// TIA Portal project "Pilot_Ultrafilter" (V20)

(* hardware
DEVICE "S7-1200 station_1"  S7-1200 Station
   slot 0: "Rack_0"  S7-1200 Rack  Rack  V1.0
   slot 1: "PLC_1"  CPU 1214C DC/DC/Rly  6ES7 214-1HG40-0XB0  V4.5
   slot 2: "AI 8x13BIT_1"  SM 1231 AI8  6ES7 231-4HF32-0XB0  V2.1
   slot 3: "AQ 2x14BIT_1"  SM 1232 AQ2  6ES7 232-4HB32-0XB0  V2.0
*)

// ===== PLC "PLC_1"  CPU 1214C DC/DC/Rly =====

VAR_GLOBAL   // PLC tag table "Default tag table"
   "IT_Pump_DryRun_Fault" AT %M0.0 : Bool;
   "IT_Pump_Wrong_Valve_Setting_fault" AT %M0.1 : Bool;
   "PID_Reset_Value" AT %M0.2 : Bool;
   "IT_EStop_NOk" AT %M0.3 : Bool;
   "ErrorBit" AT %M0.4 : Bool;   // Mindaddig amíg a hiba nem kerül nyugtázásra addig nem lehet elindítani a rendszert
   "Tag_7" AT %M0.5 : Bool;
   "Tag_8" AT %M0.6 : Bool;
   "Tag_9" AT %M0.7 : Bool;
   "Tag_10" AT %M1.0 : Bool;
   "Tag_11" AT %M1.1 : Bool;
   "Tag_12" AT %M1.2 : Bool;
   "Clock_Byte" AT %MB10 : Byte;
   "Clock_10Hz" AT %M10.0 : Bool;
   "Clock_5Hz" AT %M10.1 : Bool;
   "Clock_2.5Hz" AT %M10.2 : Bool;
   "Clock_2Hz" AT %M10.3 : Bool;
   "Clock_1.25Hz" AT %M10.4 : Bool;
   "Clock_1Hz" AT %M10.5 : Bool;
   "Clock_0.625Hz" AT %M10.6 : Bool;
   "Clock_0.5Hz" AT %M10.7 : Bool;
END_VAR

VAR_GLOBAL   // PLC tag table "Digital_Inputs"
   "DI_EStop_Ok" AT %I0.0 : Bool;   // VészStop alaphelyzetben NC
   "DI_MotorProtectionSwitch" AT %I0.1 : Bool;   // Motorvédő kapcsoló NC
   "DI_TankLevelSwitch" AT %I0.2 : Bool;   // Tartály szintjelző; Üres: 1 ; Tele:0
END_VAR

VAR_GLOBAL   // PLC tag table "Digital Outputs"
   "DO_MotorStartSign" AT %Q0.0 : Bool;
   "DO_TankFillValve" AT %Q0.1 : Bool;
   "DO_OpenPermeateValve" AT %Q0.2 : Bool;
   "DO_GreenLamp" AT %Q0.5 : Bool;
   "DO_RedLamp" AT %Q0.7 : Bool;
END_VAR

VAR_GLOBAL   // PLC tag table "Analog_Inputs"
   "AI_FT01_FlowMeter" AT %IW96 : Int;   // Szivattyú utáni áramlásmérő
   "AI_FT02_FlowMeter" AT %IW98 : Int;   // Permeátum ágban lévő áramlásmérő
   "AI_PT01_PressureTransmitter" AT %IW100 : Int;   // Membrán elötti nyomástávadó
   "AI_PT02_PressureTransmitter" AT %IW102 : Int;   // Membrán utáni nyomástávadó
END_VAR

VAR_GLOBAL   // PLC tag table "Analog_Outputs"
   "AO_PumpSpeed" AT %QW112 : Int;   // Szivattyú fordulatszámának szabályozására való analóg kimenet
END_VAR

// folder: HMI_DataBlocks

DATA_BLOCK "HMI_Inputs"   // DB4
{ S7_Optimized_Access := 'FALSE' }
VERSION : 0.1
   VAR
      "FT01_FlowMeter_l/min" : Real;
      "FT02_FlowMeter_l/min" : Real;
      PT01_PressureTransmitter_bar : Real;
      PT02_PressureTransmitter_bar : Real;
      "P01_PumpPerformance_%" : Real;
   END_VAR
BEGIN
END_DATA_BLOCK

DATA_BLOCK "HMI_Outputs"   // DB5
{ S7_Optimized_Access := 'FALSE' }
VERSION : 0.1
   VAR
      Asked_Total_Flow : Int;
      Asked_Permeate_Flow : Real;
      askedFlushingTime : DInt;
      askedVentingTime : DInt;
      "askedPumpPerformance_%" : Int;
      askedState : Int;
      askedPermeateFlowMonitoring : Bool;
      Motor_Start_Sign : Bool;
      Nyugta : Bool;
      askedGreenLight : Bool;
      askedRedLight : Bool;
      askedTankFillValveOpen : Bool;
      askedPermeateValveOpen : Bool;
   END_VAR
BEGIN
END_DATA_BLOCK

// folder: Internal_DataBlocks

DATA_BLOCK "DB_AnalogCalculatedValues"   // DB2
{ S7_Optimized_Access := 'TRUE' }
VERSION : 0.1
   VAR
      "FT01_FlowMeter_l/min" : Real;
      "FT02_FlowMeter_l/min" : Real;
      PT01_PressureTransmitter_bar : Real;
      PT02_PressureTransmitter_bar : Real;
      "P01_PumpPerformance_%" : Real;
   END_VAR
BEGIN
END_DATA_BLOCK

DATA_BLOCK "FB_ErrorHandler_DB_1"   // DB9
{ S7_Optimized_Access := 'TRUE' }
VERSION : 0.1
// stored: InstanceOfName FB_ErrorHandler
"FB_ErrorHandler"
BEGIN
END_DATA_BLOCK

DATA_BLOCK "FB_ErrorHandler_DB"   // DB10
{ S7_Optimized_Access := 'TRUE' }
VERSION : 0.1
// stored: InstanceOfName FB_ErrorHandler
"FB_ErrorHandler"
BEGIN
END_DATA_BLOCK

DATA_BLOCK "DB_StateMachine"   // DB11
{ S7_Optimized_Access := 'FALSE' }
VERSION : 0.1
   VAR
      actualState : Int;
      initState : Int := 0;
      idleState : Int := 10;
      serviceState : Int := 20;
      filteringState : Int := 100;
      filteringStateTankFilling : Int := 110;
      filteringStateVenting : Int := 120;
      filteringStateFiltering : Int := 130;
      filteringStateFlushing : Int := 140;
      filteringEnded : Int := 200;
      errorState : Int := 900;
      initState_bool : Bool;
      idleState_bool : Bool;
      serviceState_bool : Bool;
      filteringState_bool : Bool;
      filteringStateTankFilling_bool : Bool;
      filteringStateVenting_bool : Bool;
      filteringStateFiltering_bool : Bool;
      filteringStateFlushing_bool : Bool;
      filteringEnded_bool : Bool;
      errorState_bool : Bool;
   END_VAR
BEGIN
END_DATA_BLOCK

DATA_BLOCK "DB_Errors&Warnings"   // DB12
{ S7_Optimized_Access := 'FALSE' }
VERSION : 0.1
   VAR
      error : Bool;
      warning : Bool;
   END_VAR
BEGIN
END_DATA_BLOCK

DATA_BLOCK "FB_ErrorHandler_DB_2"   // DB17
{ S7_Optimized_Access := 'TRUE' }
VERSION : 0.1
// stored: InstanceOfName FB_ErrorHandler
"FB_ErrorHandler"
BEGIN
END_DATA_BLOCK

// folder: System blocks/Program resources

DATA_BLOCK "IEC_Timer_0_DB_4"   // DB13
{ S7_Optimized_Access := 'TRUE' }
AUTHOR : Simatic
FAMILY : IEC
NAME : IEC_TMR
VERSION : 1.0
// stored: InstanceOfName IEC_TIMER
"IEC_TIMER"
BEGIN
END_DATA_BLOCK

DATA_BLOCK "IEC_Timer_0_DB_5"   // DB14
{ S7_Optimized_Access := 'TRUE' }
AUTHOR : Simatic
FAMILY : IEC
NAME : IEC_TMR
VERSION : 1.0
// stored: InstanceOfName IEC_TIMER
"IEC_TIMER"
BEGIN
END_DATA_BLOCK

DATA_BLOCK "IEC_Timer_0_DB_6"   // DB15
{ S7_Optimized_Access := 'TRUE' }
AUTHOR : Simatic
FAMILY : IEC
NAME : IEC_TMR
VERSION : 1.0
// stored: InstanceOfName IEC_TIMER
"IEC_TIMER"
BEGIN
END_DATA_BLOCK

DATA_BLOCK "IEC_Timer_0_DB_7"   // DB16
{ S7_Optimized_Access := 'TRUE' }
AUTHOR : Simatic
FAMILY : IEC
NAME : IEC_TMR
VERSION : 1.0
// stored: InstanceOfName IEC_TIMER
"IEC_TIMER"
BEGIN
END_DATA_BLOCK

// folder: FC's

FUNCTION_BLOCK "FB_ErrorHandler"   // FB1, LAD
{ S7_Optimized_Access := 'TRUE' }
VERSION : 0.1
   VAR_INPUT
      startSign : Bool;
   END_VAR
   VAR
      DryRunTimer : TON_TIME;
      WrongValveSettingTimer : TON_TIME;
   END_VAR
   VAR CONSTANT
      Required_Minimum_Flow : Real := 15.0;
      Maximum_Pressure : Real := 10.0;
   END_VAR
BEGIN

REGION Network 1
   // Szárazonfutás elleni védelem
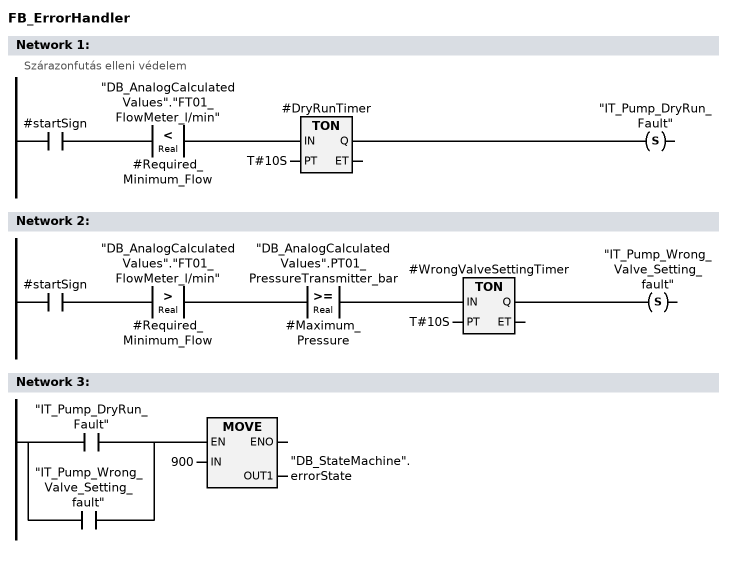
   #DryRunTimer(IN := #startSign AND ("DB_AnalogCalculatedValues"."FT01_FlowMeter_l/min" < #Required_Minimum_Flow),   // TON
                PT := T#10S);
   IF #DryRunTimer.Q THEN "IT_Pump_DryRun_Fault" := TRUE; END_IF;
END_REGION

REGION Network 2
   #WrongValveSettingTimer(IN := #startSign AND ("DB_AnalogCalculatedValues"."FT01_FlowMeter_l/min" > #Required_Minimum_Flow) AND ("DB_AnalogCalculatedValues".PT01_PressureTransmitter_bar >= #Maximum_Pressure),   // TON
                           PT := T#10S);
   IF #WrongValveSettingTimer.Q THEN "IT_Pump_Wrong_Valve_Setting_fault" := TRUE; END_IF;
END_REGION

REGION Network 3
   RUNG wire#powerrail
      Contact( "IT_Pump_DryRun_Fault" )
      wire#w1
      Move(in := 900, out1 => "DB_StateMachine".errorState)
   END_RUNG
   RUNG wire#powerrail
      Contact( "IT_Pump_Wrong_Valve_Setting_fault" )
   END_RUNG wire#w1
   // the same network as SCL:
   IF "IT_Pump_DryRun_Fault" OR "IT_Pump_Wrong_Valve_Setting_fault" THEN
       "DB_StateMachine".errorState := 900;
   END_IF;
END_REGION
END_FUNCTION_BLOCK

FUNCTION "FC_AnalogInputScale" : Void   // FC1, LAD
{ S7_Optimized_Access := 'TRUE' }
VERSION : 0.1
   VAR_INPUT
      InputAnalogValue : Int;
      MinimumAnalogValue : Int;
      MaximumAnalogValue : Int;
      MinimumScaledValue : Real;
      MaxmimumScaledValue : Int;
   END_VAR
   VAR_OUTPUT
      OutputScaledValue : Real;
   END_VAR
   VAR_TEMP
      NormalizedValue : Real;
   END_VAR
BEGIN

REGION Network 1
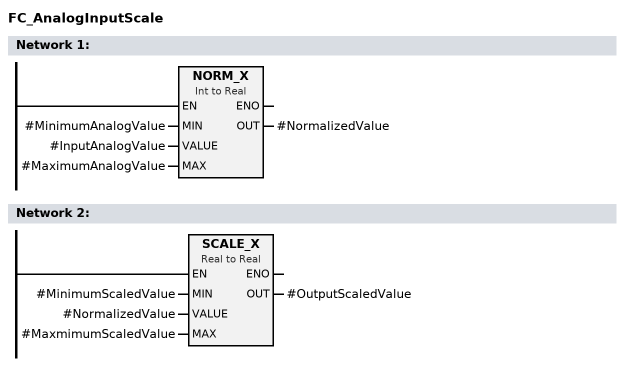
   RUNG wire#powerrail
      { S7_Templates := "[SrcType := Int, DestType := Real]" } Normalize(min := #MinimumAnalogValue, value := #InputAnalogValue, max := #MaximumAnalogValue, out => #NormalizedValue)
   END_RUNG
   // the same network as SCL:
   #NormalizedValue := NORM_X(MIN := #MinimumAnalogValue, VALUE := #InputAnalogValue, MAX := #MaximumAnalogValue);
END_REGION

REGION Network 2
   RUNG wire#powerrail
      { S7_Templates := "[SrcType := Real, DestType := Real]" } Scale(min := #MinimumScaledValue, value := #NormalizedValue, max := #MaxmimumScaledValue, out => #OutputScaledValue)
   END_RUNG
   // the same network as SCL:
   #OutputScaledValue := SCALE_X(MIN := #MinimumScaledValue, VALUE := #NormalizedValue, MAX := #MaxmimumScaledValue);
END_REGION
END_FUNCTION

FUNCTION "FC_ProcessAnalogInputs" : Void   // FC2, LAD
{ S7_Optimized_Access := 'TRUE' }
VERSION : 0.1
   VAR CONSTANT
      FT01_MinimumAnalogValue : Int := 1659;   // Minimális analóg érték a szivattyú utáni áramlásmérő által
      FT02_MinimumAnalogValue : Int := 1382;   // Minimális analóg érték a permeátum ágban lévő áramlásmérőnél
      "PT01-02_MinimumAnalogValue" : Int := 0;   // Minimális analóg érték a két nyomástávadónál
      ALL_MaximumAnalogValue : Int := 27648;   // Maximális analóg érték, összesnél megegyezik
      FT01_MinimumFlowValue : Real := 9.0;   // Legkisebb áramlás amit a szivattyú utáni áramlásmérő tud
      FT02_MinimumFlowValue : Real := 0.5;   // Legkisebb áramlás amit a permeátum ágban lévő áramlásmérő mérni tud
      FT01_MaximumFlowValue : Int := 150;   // Legnagyobb áramlás amit a szivattyú utáni áramlásmérő tud
      FT02_MaximumFlowValue : Int := 10;   // Legnagyobb áramlás amit a premátum ágban lévő áramlásmérő tud
      "PT01-02_MinimumPressureValue" : Real := 0.0;   // Legkisebb nyomás amit a nyomástávadók tudnak
      "PT01-02MaximumPressureValue" : Int := 10;   // Legnagyobb nyomás amit a nyomástávadók tudnak
   END_VAR
   VAR_TEMP   // added for the SCL form of the ladder/FBD networks
      _w1 : Bool;
   END_VAR
BEGIN

REGION Network 1
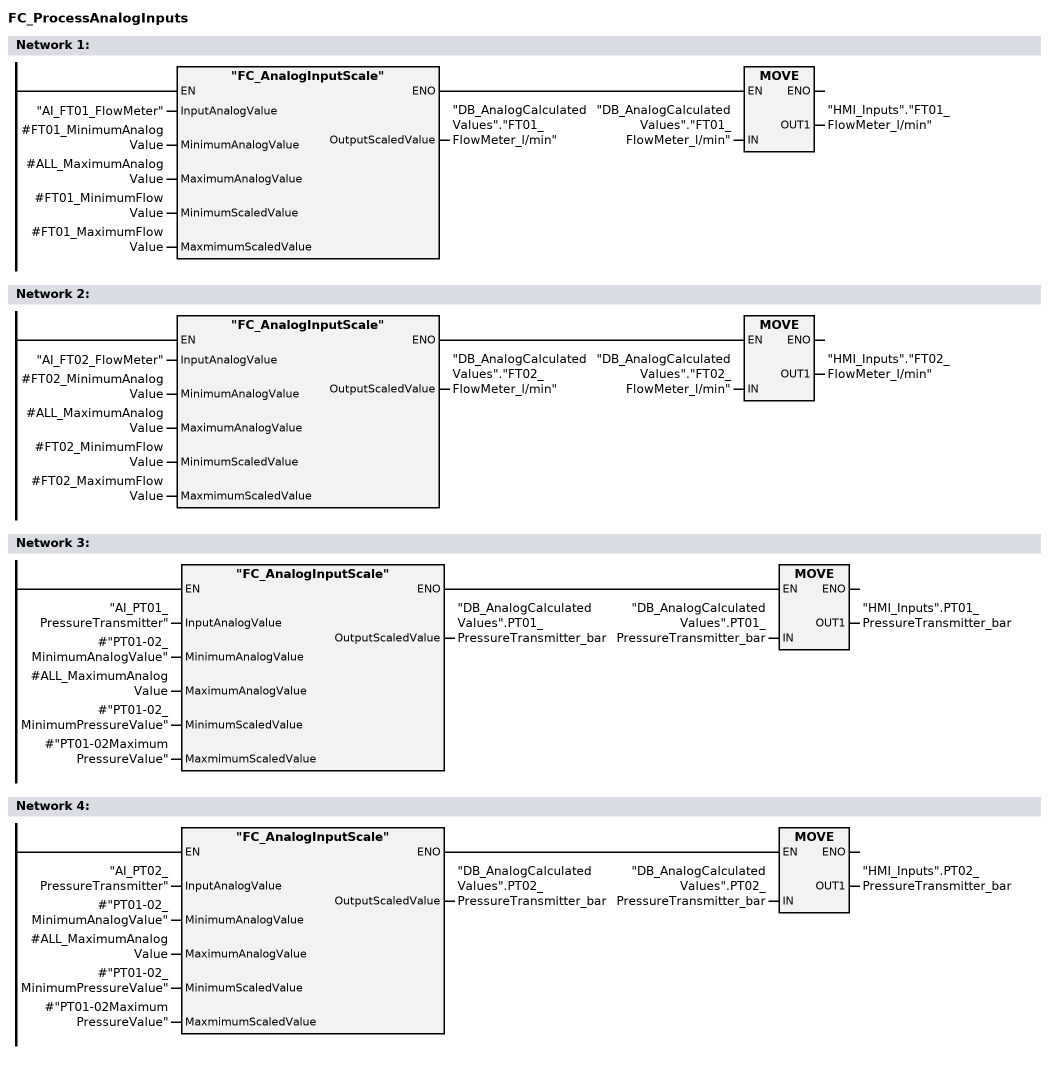
   RUNG wire#powerrail
      "FC_AnalogInputScale"(InputAnalogValue := "AI_FT01_FlowMeter", MinimumAnalogValue := #FT01_MinimumAnalogValue, MaximumAnalogValue := #ALL_MaximumAnalogValue, MinimumScaledValue := #FT01_MinimumFlowValue, MaxmimumScaledValue := #FT01_MaximumFlowValue, OutputScaledValue => "DB_AnalogCalculatedValues"."FT01_FlowMeter_l/min")
      Move(in := "DB_AnalogCalculatedValues"."FT01_FlowMeter_l/min", out1 => "HMI_Inputs"."FT01_FlowMeter_l/min")
   END_RUNG
   // the same network as SCL:
   "FC_AnalogInputScale"(InputAnalogValue := "AI_FT01_FlowMeter",
                         MinimumAnalogValue := #FT01_MinimumAnalogValue,
                         MaximumAnalogValue := #ALL_MaximumAnalogValue,
                         MinimumScaledValue := #FT01_MinimumFlowValue,
                         MaxmimumScaledValue := #FT01_MaximumFlowValue,
                         OutputScaledValue => "DB_AnalogCalculatedValues"."FT01_FlowMeter_l/min",
                         ENO => #_w1);
   IF #_w1 THEN
       "HMI_Inputs"."FT01_FlowMeter_l/min" := "DB_AnalogCalculatedValues"."FT01_FlowMeter_l/min";
   END_IF;
END_REGION

REGION Network 2
   RUNG wire#powerrail
      "FC_AnalogInputScale"(InputAnalogValue := "AI_FT02_FlowMeter", MinimumAnalogValue := #FT02_MinimumAnalogValue, MaximumAnalogValue := #ALL_MaximumAnalogValue, MinimumScaledValue := #FT02_MinimumFlowValue, MaxmimumScaledValue := #FT02_MaximumFlowValue, OutputScaledValue => "DB_AnalogCalculatedValues"."FT02_FlowMeter_l/min")
      Move(in := "DB_AnalogCalculatedValues"."FT02_FlowMeter_l/min", out1 => "HMI_Inputs"."FT02_FlowMeter_l/min")
   END_RUNG
   // the same network as SCL:
   "FC_AnalogInputScale"(InputAnalogValue := "AI_FT02_FlowMeter",
                         MinimumAnalogValue := #FT02_MinimumAnalogValue,
                         MaximumAnalogValue := #ALL_MaximumAnalogValue,
                         MinimumScaledValue := #FT02_MinimumFlowValue,
                         MaxmimumScaledValue := #FT02_MaximumFlowValue,
                         OutputScaledValue => "DB_AnalogCalculatedValues"."FT02_FlowMeter_l/min",
                         ENO => #_w1);
   IF #_w1 THEN
       "HMI_Inputs"."FT02_FlowMeter_l/min" := "DB_AnalogCalculatedValues"."FT02_FlowMeter_l/min";
   END_IF;
END_REGION

REGION Network 3
   RUNG wire#powerrail
      "FC_AnalogInputScale"(InputAnalogValue := "AI_PT01_PressureTransmitter", MinimumAnalogValue := #"PT01-02_MinimumAnalogValue", MaximumAnalogValue := #ALL_MaximumAnalogValue, MinimumScaledValue := #"PT01-02_MinimumPressureValue", MaxmimumScaledValue := #"PT01-02MaximumPressureValue", OutputScaledValue => "DB_AnalogCalculatedValues".PT01_PressureTransmitter_bar)
      Move(in := "DB_AnalogCalculatedValues".PT01_PressureTransmitter_bar, out1 => "HMI_Inputs".PT01_PressureTransmitter_bar)
   END_RUNG
   // the same network as SCL:
   "FC_AnalogInputScale"(InputAnalogValue := "AI_PT01_PressureTransmitter",
                         MinimumAnalogValue := #"PT01-02_MinimumAnalogValue",
                         MaximumAnalogValue := #ALL_MaximumAnalogValue,
                         MinimumScaledValue := #"PT01-02_MinimumPressureValue",
                         MaxmimumScaledValue := #"PT01-02MaximumPressureValue",
                         OutputScaledValue => "DB_AnalogCalculatedValues".PT01_PressureTransmitter_bar,
                         ENO => #_w1);
   IF #_w1 THEN
       "HMI_Inputs".PT01_PressureTransmitter_bar := "DB_AnalogCalculatedValues".PT01_PressureTransmitter_bar;
   END_IF;
END_REGION

REGION Network 4
   RUNG wire#powerrail
      "FC_AnalogInputScale"(InputAnalogValue := "AI_PT02_PressureTransmitter", MinimumAnalogValue := #"PT01-02_MinimumAnalogValue", MaximumAnalogValue := #ALL_MaximumAnalogValue, MinimumScaledValue := #"PT01-02_MinimumPressureValue", MaxmimumScaledValue := #"PT01-02MaximumPressureValue", OutputScaledValue => "DB_AnalogCalculatedValues".PT02_PressureTransmitter_bar)
      Move(in := "DB_AnalogCalculatedValues".PT02_PressureTransmitter_bar, out1 => "HMI_Inputs".PT02_PressureTransmitter_bar)
   END_RUNG
   // the same network as SCL:
   "FC_AnalogInputScale"(InputAnalogValue := "AI_PT02_PressureTransmitter",
                         MinimumAnalogValue := #"PT01-02_MinimumAnalogValue",
                         MaximumAnalogValue := #ALL_MaximumAnalogValue,
                         MinimumScaledValue := #"PT01-02_MinimumPressureValue",
                         MaxmimumScaledValue := #"PT01-02MaximumPressureValue",
                         OutputScaledValue => "DB_AnalogCalculatedValues".PT02_PressureTransmitter_bar,
                         ENO => #_w1);
   IF #_w1 THEN
       "HMI_Inputs".PT02_PressureTransmitter_bar := "DB_AnalogCalculatedValues".PT02_PressureTransmitter_bar;
   END_IF;
END_REGION
END_FUNCTION

FUNCTION "FC_IdleState" : Void   // FC3, SCL
{ S7_Optimized_Access := 'TRUE' }
VERSION : 0.1
BEGIN
   "DO_MotorStartSign" := FALSE;
   "DO_TankFillValve" := FALSE;
   "DO_OpenPermeateValve" := FALSE;
   "DO_GreenLamp" := FALSE;
   "DO_RedLamp" := FALSE;
   "AO_PumpSpeed" := 0;
END_FUNCTION

FUNCTION "FC_TankFilling" : Void   // FC4, LAD
{ S7_Optimized_Access := 'TRUE' }
VERSION : 0.1
BEGIN

REGION Network 1
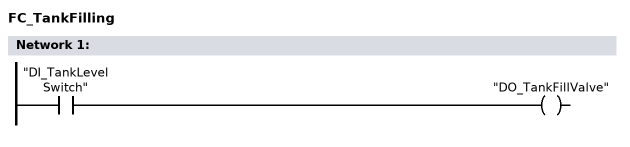
   RUNG wire#powerrail
      Contact( "DI_TankLevelSwitch" )
      Coil( "DO_TankFillValve" )
   END_RUNG
   // the same network as SCL:
   "DO_TankFillValve" := "DI_TankLevelSwitch";
END_REGION
END_FUNCTION

FUNCTION "FC_Membrane_FlushState" : Void   // FC5, LAD
{ S7_Optimized_Access := 'TRUE' }
VERSION : 0.1
   VAR_OUTPUT
      flushingOver : Bool;
      successfullFlushing : Bool;
   END_VAR
   VAR_TEMP
      flushingOverTemp : Bool;
   END_VAR
BEGIN

REGION Network 1
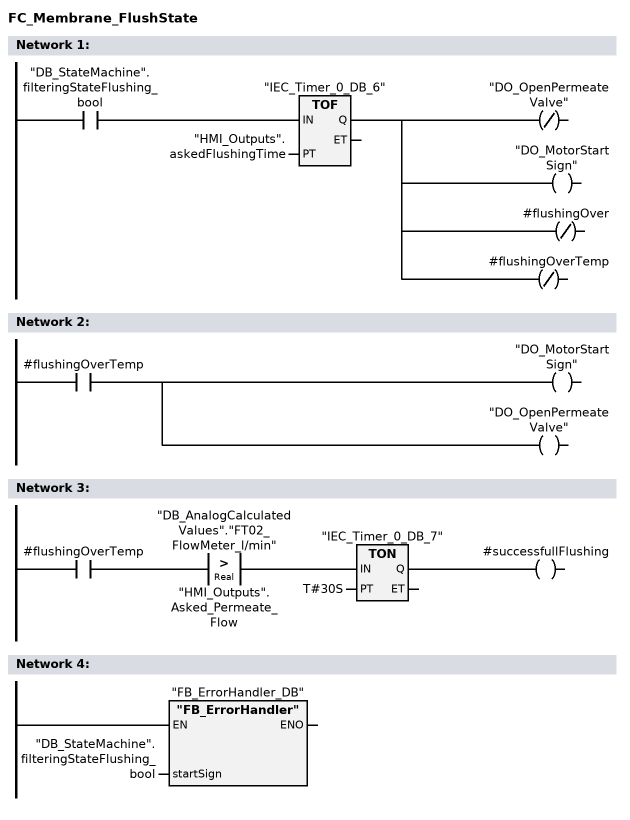
   "IEC_Timer_0_DB_6".TOF(IN := "DB_StateMachine".filteringStateFlushing_bool,
                          PT := "HMI_Outputs".askedFlushingTime);
   "DO_OpenPermeateValve" := NOT "IEC_Timer_0_DB_6".Q;
   "DO_MotorStartSign" := "IEC_Timer_0_DB_6".Q;
   #flushingOver := NOT "IEC_Timer_0_DB_6".Q;
   #flushingOverTemp := NOT "IEC_Timer_0_DB_6".Q;
END_REGION

REGION Network 2
   RUNG wire#powerrail
      Contact( #flushingOverTemp )
      wire#w1
      Coil( "DO_MotorStartSign" )
   END_RUNG
   RUNG wire#w1
      Coil( "DO_OpenPermeateValve" )
   END_RUNG
   // the same network as SCL:
   "DO_MotorStartSign" := #flushingOverTemp;
   "DO_OpenPermeateValve" := #flushingOverTemp;
END_REGION

REGION Network 3
   "IEC_Timer_0_DB_7".TON(IN := #flushingOverTemp AND ("DB_AnalogCalculatedValues"."FT02_FlowMeter_l/min" > "HMI_Outputs".Asked_Permeate_Flow),
                          PT := T#30S);
   #successfullFlushing := "IEC_Timer_0_DB_7".Q;
END_REGION

REGION Network 4
   RUNG wire#powerrail
      "FB_ErrorHandler_DB"(startSign := "DB_StateMachine".filteringStateFlushing_bool)
   END_RUNG
   // the same network as SCL:
   "FB_ErrorHandler_DB"(startSign := "DB_StateMachine".filteringStateFlushing_bool);   // "FB_ErrorHandler"
END_REGION
END_FUNCTION

FUNCTION "FC_ServiceState" : Void   // FC6, LAD
{ S7_Optimized_Access := 'TRUE' }
VERSION : 0.1
// manuális szervíz állás, minden paraméter a HMI ről állítható
BEGIN

REGION Network 1
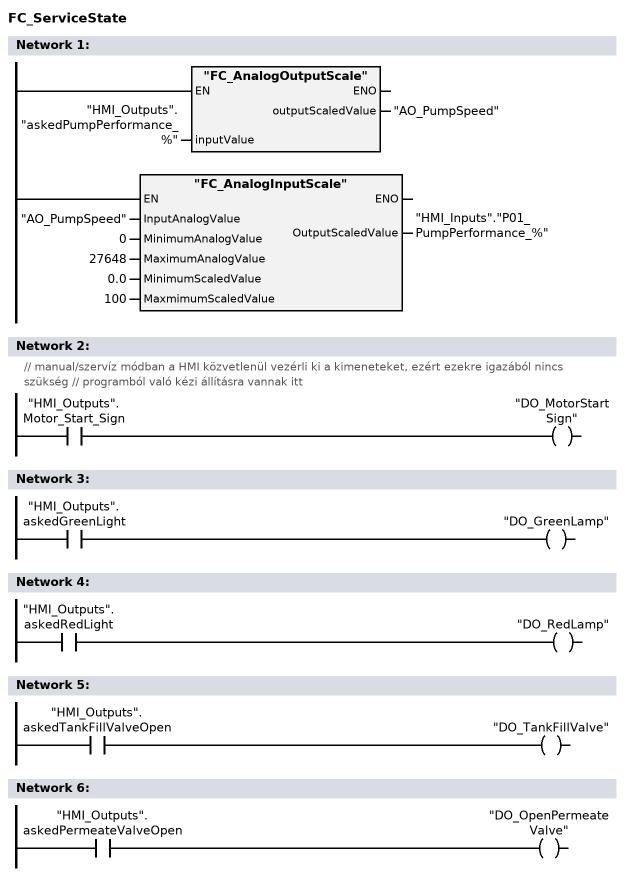
   RUNG wire#powerrail
      "FC_AnalogOutputScale"(inputValue := "HMI_Outputs"."askedPumpPerformance_%", outputScaledValue => "AO_PumpSpeed")
   END_RUNG
   RUNG wire#powerrail
      "FC_AnalogInputScale"(InputAnalogValue := "AO_PumpSpeed", MinimumAnalogValue := 0, MaximumAnalogValue := 27648, MinimumScaledValue := 0.0, MaxmimumScaledValue := 100, OutputScaledValue => "HMI_Inputs"."P01_PumpPerformance_%")
   END_RUNG
   // the same network as SCL:
   "FC_AnalogOutputScale"(inputValue := "HMI_Outputs"."askedPumpPerformance_%",
                          outputScaledValue => "AO_PumpSpeed");
   "FC_AnalogInputScale"(InputAnalogValue := "AO_PumpSpeed",
                         MinimumAnalogValue := 0,
                         MaximumAnalogValue := 27648,
                         MinimumScaledValue := 0.0,
                         MaxmimumScaledValue := 100,
                         OutputScaledValue => "HMI_Inputs"."P01_PumpPerformance_%");
END_REGION

REGION Network 2
   // // manual/szervíz módban a HMI közvetlenül vezérli ki a kimeneteket, ezért ezekre igazából nincs szükség // programból való kézi állításra vannak itt
   RUNG wire#powerrail
      Contact( "HMI_Outputs".Motor_Start_Sign )
      Coil( "DO_MotorStartSign" )
   END_RUNG
   // the same network as SCL:
   "DO_MotorStartSign" := "HMI_Outputs".Motor_Start_Sign;
END_REGION

REGION Network 3
   RUNG wire#powerrail
      Contact( "HMI_Outputs".askedGreenLight )
      Coil( "DO_GreenLamp" )
   END_RUNG
   // the same network as SCL:
   "DO_GreenLamp" := "HMI_Outputs".askedGreenLight;
END_REGION

REGION Network 4
   RUNG wire#powerrail
      Contact( "HMI_Outputs".askedRedLight )
      Coil( "DO_RedLamp" )
   END_RUNG
   // the same network as SCL:
   "DO_RedLamp" := "HMI_Outputs".askedRedLight;
END_REGION

REGION Network 5
   RUNG wire#powerrail
      Contact( "HMI_Outputs".askedTankFillValveOpen )
      Coil( "DO_TankFillValve" )
   END_RUNG
   // the same network as SCL:
   "DO_TankFillValve" := "HMI_Outputs".askedTankFillValveOpen;
END_REGION

REGION Network 6
   RUNG wire#powerrail
      Contact( "HMI_Outputs".askedPermeateValveOpen )
      Coil( "DO_OpenPermeateValve" )
   END_RUNG
   // the same network as SCL:
   "DO_OpenPermeateValve" := "HMI_Outputs".askedPermeateValveOpen;
END_REGION
END_FUNCTION

FUNCTION "FC_AnalogOutputScale" : Void   // FC7, LAD
{ S7_Optimized_Access := 'TRUE' }
VERSION : 0.1
   VAR_INPUT
      inputValue : Real;
   END_VAR
   VAR_OUTPUT
      outputScaledValue : Int;
   END_VAR
   VAR_TEMP
      normalizedValue : Real;
   END_VAR
BEGIN

REGION Network 1
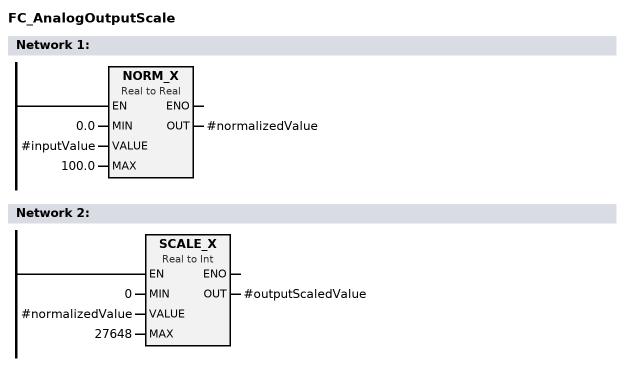
   RUNG wire#powerrail
      { S7_Templates := "[SrcType := Real, DestType := Real]" } Normalize(min := 0.0, value := #inputValue, max := 100.0, out => #normalizedValue)
   END_RUNG
   // the same network as SCL:
   #normalizedValue := NORM_X(MIN := 0.0, VALUE := #inputValue, MAX := 100.0);
END_REGION

REGION Network 2
   RUNG wire#powerrail
      { S7_Templates := "[SrcType := Real, DestType := Int]" } Scale(min := 0, value := #normalizedValue, max := 27648, out => #outputScaledValue)
   END_RUNG
   // the same network as SCL:
   #outputScaledValue := SCALE_X(MIN := 0, VALUE := #normalizedValue, MAX := 27648);
END_REGION
END_FUNCTION

FUNCTION "FC_VentingMembraneState" : Void   // FC8, LAD
{ S7_Optimized_Access := 'TRUE' }
VERSION : 0.1
   VAR_INPUT
      askedVentingTime : DInt;
   END_VAR
   VAR_OUTPUT
      ventingOver : Bool;
   END_VAR
   VAR_TEMP   // added for the SCL form of the ladder/FBD networks
      _w1 : Bool;
   END_VAR
BEGIN

REGION Network 1
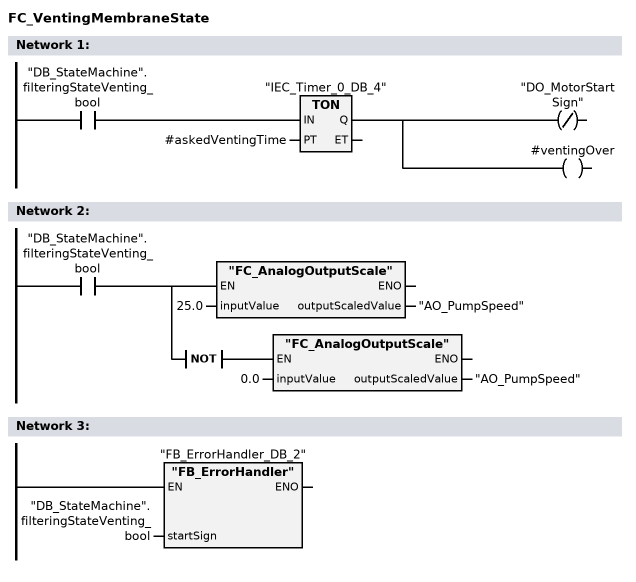
   "IEC_Timer_0_DB_4".TON(IN := "DB_StateMachine".filteringStateVenting_bool, PT := #askedVentingTime);
   "DO_MotorStartSign" := NOT "IEC_Timer_0_DB_4".Q;
   #ventingOver := "IEC_Timer_0_DB_4".Q;
END_REGION

REGION Network 2
   RUNG wire#powerrail
      Contact( "DB_StateMachine".filteringStateVenting_bool )
      wire#w1
      "FC_AnalogOutputScale"(inputValue := 25.0, outputScaledValue => "AO_PumpSpeed")
   END_RUNG
   RUNG wire#w1
      Not()
      "FC_AnalogOutputScale"(inputValue := 0.0, outputScaledValue => "AO_PumpSpeed")
   END_RUNG
   // the same network as SCL:
   #_w1 := "DB_StateMachine".filteringStateVenting_bool;
   IF #_w1 THEN "FC_AnalogOutputScale"(inputValue := 25.0, outputScaledValue => "AO_PumpSpeed"); END_IF;
   IF NOT #_w1 THEN "FC_AnalogOutputScale"(inputValue := 0.0, outputScaledValue => "AO_PumpSpeed"); END_IF;
END_REGION

REGION Network 3
   RUNG wire#powerrail
      "FB_ErrorHandler_DB_2"(startSign := "DB_StateMachine".filteringStateVenting_bool)
   END_RUNG
   // the same network as SCL:
   "FB_ErrorHandler_DB_2"(startSign := "DB_StateMachine".filteringStateVenting_bool);   // "FB_ErrorHandler"
END_REGION
END_FUNCTION

FUNCTION "FC_FilteringState" : Void   // FC9, LAD
{ S7_Optimized_Access := 'TRUE' }
VERSION : 0.1
   VAR_OUTPUT
      minimumPermeateFlowReached : Bool;
   END_VAR
   VAR_TEMP
      stateSwitching : Bool;
   END_VAR
BEGIN

REGION Network 1
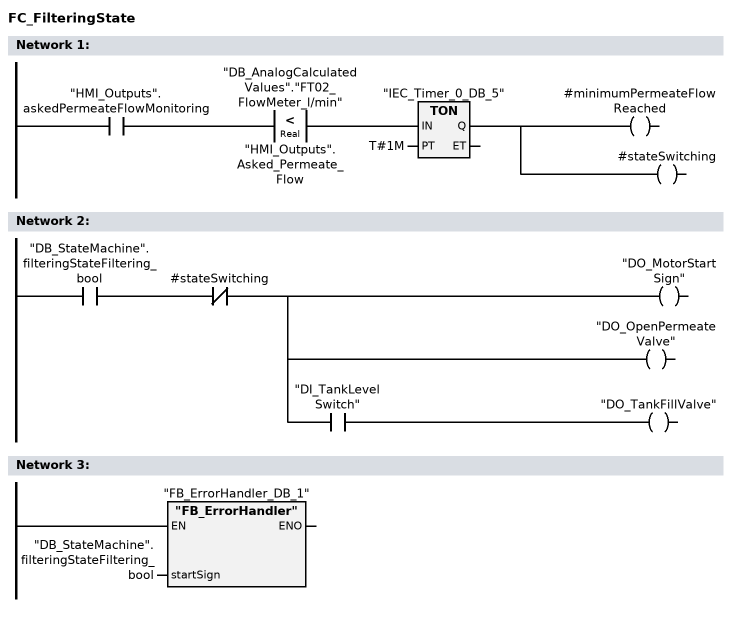
   "IEC_Timer_0_DB_5".TON(IN := "HMI_Outputs".askedPermeateFlowMonitoring AND ("DB_AnalogCalculatedValues"."FT02_FlowMeter_l/min" < "HMI_Outputs".Asked_Permeate_Flow),
                          PT := T#1M);
   #minimumPermeateFlowReached := "IEC_Timer_0_DB_5".Q;
   #stateSwitching := "IEC_Timer_0_DB_5".Q;
END_REGION

REGION Network 2
   RUNG wire#powerrail
      Contact( "DB_StateMachine".filteringStateFiltering_bool )
      I_Contact( #stateSwitching )
      wire#w1
      Coil( "DO_MotorStartSign" )
   END_RUNG
   RUNG wire#w1
      Coil( "DO_OpenPermeateValve" )
   END_RUNG
   RUNG wire#w1
      Contact( "DI_TankLevelSwitch" )
      Coil( "DO_TankFillValve" )
   END_RUNG
   // the same network as SCL:
   "DO_MotorStartSign" := "DB_StateMachine".filteringStateFiltering_bool AND NOT #stateSwitching;
   "DO_OpenPermeateValve" := "DO_MotorStartSign";
   "DO_TankFillValve" := "DO_MotorStartSign" AND "DI_TankLevelSwitch";
END_REGION

REGION Network 3
   RUNG wire#powerrail
      "FB_ErrorHandler_DB_1"(startSign := "DB_StateMachine".filteringStateFiltering_bool)
   END_RUNG
   // the same network as SCL:
   "FB_ErrorHandler_DB_1"(startSign := "DB_StateMachine".filteringStateFiltering_bool);   // "FB_ErrorHandler"
END_REGION
END_FUNCTION

FUNCTION "FC_FilteringEndedState" : Void   // FC10, LAD
{ S7_Optimized_Access := 'TRUE' }
VERSION : 0.1
BEGIN

REGION Network 1
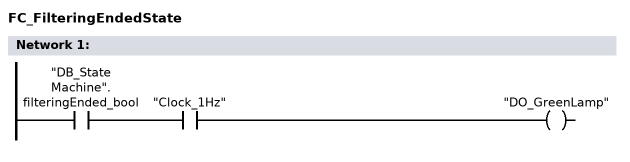
   RUNG wire#powerrail
      Contact( "DB_StateMachine".filteringEnded_bool )
      Contact( "Clock_1Hz" )
      Coil( "DO_GreenLamp" )
   END_RUNG
   // the same network as SCL:
   "DO_GreenLamp" := "DB_StateMachine".filteringEnded_bool AND "Clock_1Hz";
END_REGION

REGION Network 2 (SCL)
   WHILE "DB_StateMachine".filteringEnded_bool DO

       // Statement section WHILE
       "DO_MotorStartSign" := FALSE;
       "DO_TankFillValve" := FALSE;
       "DO_OpenPermeateValve" := FALSE;
       "DO_RedLamp" := FALSE;
       ;
   END_WHILE;
END_REGION
END_FUNCTION

FUNCTION "FC_ErrorState" : Void   // FC11, LAD
{ S7_Optimized_Access := 'TRUE' }
VERSION : 0.1
BEGIN

REGION Network 1
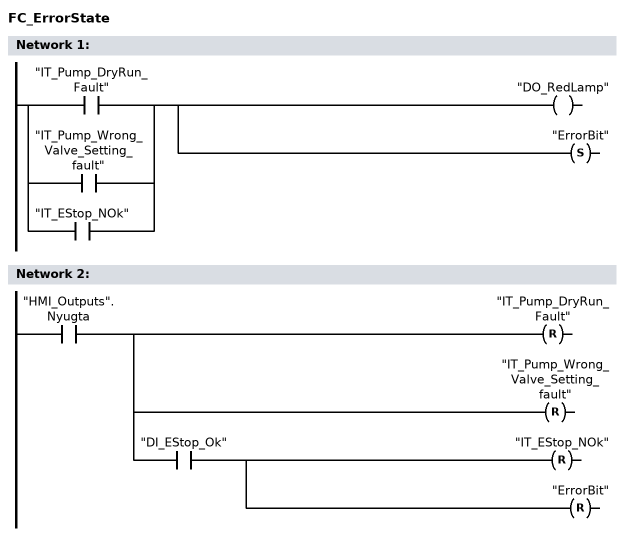
   RUNG wire#powerrail
      Contact( "IT_Pump_DryRun_Fault" )
      wire#w1
      Coil( "DO_RedLamp" )
   END_RUNG
   RUNG wire#powerrail
      Contact( "IT_Pump_Wrong_Valve_Setting_fault" )
   END_RUNG wire#w1
   RUNG wire#powerrail
      Contact( "IT_EStop_NOk" )
   END_RUNG wire#w1
   RUNG wire#w1
      S_Coil( "ErrorBit" )
   END_RUNG
   // the same network as SCL:
   "DO_RedLamp" := "IT_Pump_DryRun_Fault" OR "IT_Pump_Wrong_Valve_Setting_fault" OR "IT_EStop_NOk";
   IF "DO_RedLamp" THEN "ErrorBit" := TRUE; END_IF;
END_REGION

REGION Network 2
   RUNG wire#powerrail
      Contact( "HMI_Outputs".Nyugta )
      wire#w1
      R_Coil( "IT_Pump_DryRun_Fault" )
   END_RUNG
   RUNG wire#w1
      R_Coil( "IT_Pump_Wrong_Valve_Setting_fault" )
   END_RUNG
   RUNG wire#w1
      Contact( "DI_EStop_Ok" )
      wire#w2
      R_Coil( "IT_EStop_NOk" )
   END_RUNG
   RUNG wire#w2
      R_Coil( "ErrorBit" )
   END_RUNG
   // the same network as SCL:
   IF "HMI_Outputs".Nyugta THEN
       "IT_Pump_DryRun_Fault" := FALSE;
       "IT_Pump_Wrong_Valve_Setting_fault" := FALSE;
   END_IF;
   IF "HMI_Outputs".Nyugta AND "DI_EStop_Ok" THEN
       "IT_EStop_NOk" := FALSE;
       "ErrorBit" := FALSE;
   END_IF;
END_REGION

REGION Network 4 (SCL)
   "DB_StateMachine".initState_bool := FALSE;
   "DB_StateMachine".idleState_bool := FALSE;
   "DB_StateMachine".serviceState_bool := FALSE;
   "DB_StateMachine".filteringState_bool := FALSE;
   "DB_StateMachine".filteringStateTankFilling_bool := FALSE;
   "DB_StateMachine".filteringStateVenting_bool := FALSE;
   "DB_StateMachine".filteringStateFiltering_bool := FALSE;
   "DB_StateMachine".filteringStateFlushing_bool := FALSE;
   "DB_StateMachine".filteringEnded_bool := FALSE;

   "DB_StateMachine".errorState_bool := TRUE;
END_REGION
END_FUNCTION

// folder: OB's

ORGANIZATION_BLOCK "Main"   // OB1, LAD, ProgramCycle
TITLE = "Main Program Sweep (Cycle)"
{ S7_Optimized_Access := 'TRUE' }
VERSION : 0.1
   VAR_INPUT
      Initial_Call : Bool;   // Initial call of this OB
      Remanence : Bool;   // =True, if remanent data are available
   END_VAR
   VAR_TEMP
      ventingOver : Bool;
      minimumPermeateFlowReached : Bool;
      flushingOver : Bool;
      successfullFlushing : Bool;
   END_VAR
   VAR CONSTANT
      Helper : Int;
   END_VAR
BEGIN

REGION Network 1 (SCL)
   CASE "DB_StateMachine".actualState OF

       10:  // idle állapot, ahol a kimenetek nullázva vannak 

           "DB_StateMachine".idleState_bool:= TRUE;
           "FC_IdleState"();
           IF NOT "ErrorBit" THEN
               // ha nincs hiba és indítási jelet kapunk akkor mehet a kívánt "state"
               "DB_StateMachine".actualState := "HMI_Outputs".askedState;
               "DB_StateMachine".idleState_bool := FALSE;
               ;
           END_IF;


           ;
       20:  // manuális szervíz állás, minden paraméter a HMI ről állítható

           "DB_StateMachine".serviceState_bool := TRUE;
           "FC_ServiceState"();
           "DB_StateMachine".actualState := "HMI_Outputs".askedState;

           //false ág nincs a statenek, mert az a HMI ről lesz átállítva

           ;
       100:  // nincs rá szükség
           ;
       110:  // tartály feltöltő állás, addig fut amig a tartály nincs tele

           "DB_StateMachine".filteringStateTankFilling_bool := TRUE;
           "FC_TankFilling"();



           IF NOT "DO_TankFillValve" THEN
               "DB_StateMachine".actualState := 120;
               "DB_StateMachine".filteringStateTankFilling_bool := FALSE;
               ;
           END_IF;

           IF NOT "HMI_Outputs".Motor_Start_Sign THEN

               "DB_StateMachine".actualState := "HMI_Outputs".askedState;
               "DB_StateMachine".filteringStateTankFilling_bool := FALSE;
               ;
           END_IF;

           ;
       120:  // légtelenítési fázis a megadott ideig 

           "DB_StateMachine".filteringStateVenting_bool := TRUE;

           "FC_VentingMembraneState"
           (
            askedVentingTime := "HMI_Outputs".askedVentingTime,
               ventingOver => #ventingOver
           );
           IF #ventingOver THEN
               "DB_StateMachine".actualState := 130;
               "DB_StateMachine".filteringStateVenting_bool := FALSE;
               ;

           END_IF;
           IF NOT "HMI_Outputs".Motor_Start_Sign THEN

               "DB_StateMachine".actualState := "HMI_Outputs".askedState;
               "DB_StateMachine".filteringStateVenting_bool := FALSE;
               ;
           END_IF;

           ;
       130:  // szűrési állapot, a pid vezérlő állítja a térfogatáramot

           "DB_StateMachine".filteringStateFiltering_bool := TRUE;

           "FC_FilteringState"
           (
            minimumPermeateFlowReached => #minimumPermeateFlowReached
           );

           IF #minimumPermeateFlowReached THEN

               "DB_StateMachine".actualState := 140;
               "DB_StateMachine".filteringStateFiltering_bool := FALSE;
               ;
           END_IF;
           IF NOT "HMI_Outputs".Motor_Start_Sign THEN

               "DB_StateMachine".actualState := "HMI_Outputs".askedState;
               "DB_StateMachine".filteringStateFiltering_bool := FALSE;
               ;
           END_IF;

           ;
       140:  // membrán öblítési fázis, HMI-n beállított ideig tart

           "DB_StateMachine".filteringStateFlushing_bool := TRUE;

           "FC_Membrane_FlushState"
           (
            flushingOver => #flushingOver,
            successfullFlushing => #successfullFlushing
           );

           IF #flushingOver AND #successfullFlushing THEN

               "DB_StateMachine".actualState := 130;
               "DB_StateMachine".filteringStateFlushing_bool := FALSE;
               ;
           ELSIF #flushingOver AND NOT #successfullFlushing THEN

               "DB_StateMachine".actualState := 200;
               "DB_StateMachine".filteringStateFlushing_bool := FALSE;
           END_IF;

           IF NOT "HMI_Outputs".Motor_Start_Sign THEN

               "DB_StateMachine".actualState := "HMI_Outputs".askedState;
               "DB_StateMachine".filteringStateFiltering_bool := FALSE;
               ;
           END_IF;

           ;
       200:  // Statement section case 2 to 4

           "DB_StateMachine".filteringEnded_bool := TRUE;
           "FC_FilteringEndedState"();

           IF "HMI_Outputs".Nyugta THEN

               "DB_StateMachine".actualState := 10;
               "DB_StateMachine".filteringEnded_bool := FALSE;
               ;
           END_IF;

           ;
       900:  // hibaállapot, hiba megszűnése és nyugtázás esetén az idle állapotba kerülünk

           "DB_StateMachine".errorState_bool := TRUE;
           "ErrorBit" := TRUE;
           "FC_ErrorState"();

           IF NOT "ErrorBit" THEN

               "DB_StateMachine".actualState := 10;
               "DB_StateMachine".errorState_bool := FALSE;
               ;
           END_IF;

           ;
       ELSE  // Statement section ELSE
           ;
   END_CASE;
END_REGION

REGION Network 2
   // Az összes analóg bemenetre kiszámolja az értékeket SI mértékegységben és a DB_analogCalculatedValues táblába helyezi.
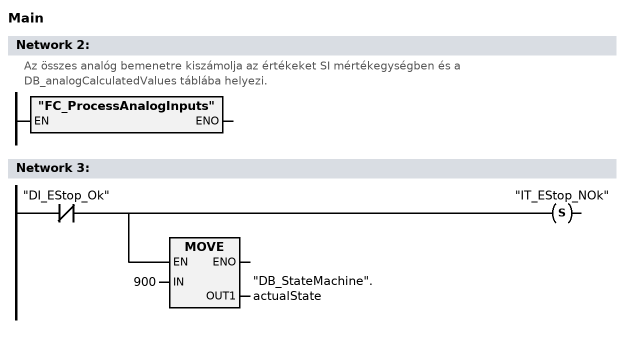
   RUNG wire#powerrail
      "FC_ProcessAnalogInputs"()
   END_RUNG
   // the same network as SCL:
   "FC_ProcessAnalogInputs"();
END_REGION

REGION Network 3
   RUNG wire#powerrail
      I_Contact( "DI_EStop_Ok" )
      wire#w1
      S_Coil( "IT_EStop_NOk" )
   END_RUNG
   RUNG wire#w1
      Move(in := 900, out1 => "DB_StateMachine".actualState)
   END_RUNG
   // the same network as SCL:
   IF NOT "DI_EStop_Ok" THEN
       "IT_EStop_NOk" := TRUE;
       "DB_StateMachine".actualState := 900;
   END_IF;
END_REGION
END_ORGANIZATION_BLOCK

ORGANIZATION_BLOCK "CyclicInterrupt"   // OB30, LAD, CyclicInterrupt
{ S7_Optimized_Access := 'TRUE' }
VERSION : 0.1
   VAR_INPUT
      Initial_Call : Bool;   // Initial call of this OB
      Event_Count : Int;   // Events discarded
   END_VAR
   VAR_TEMP
      Required_Flow : Real;
      Actual_Flow : Real;
      Ramped_Required_Flow : Real;
      pidMode : Int;
   END_VAR
BEGIN

REGION Network 1
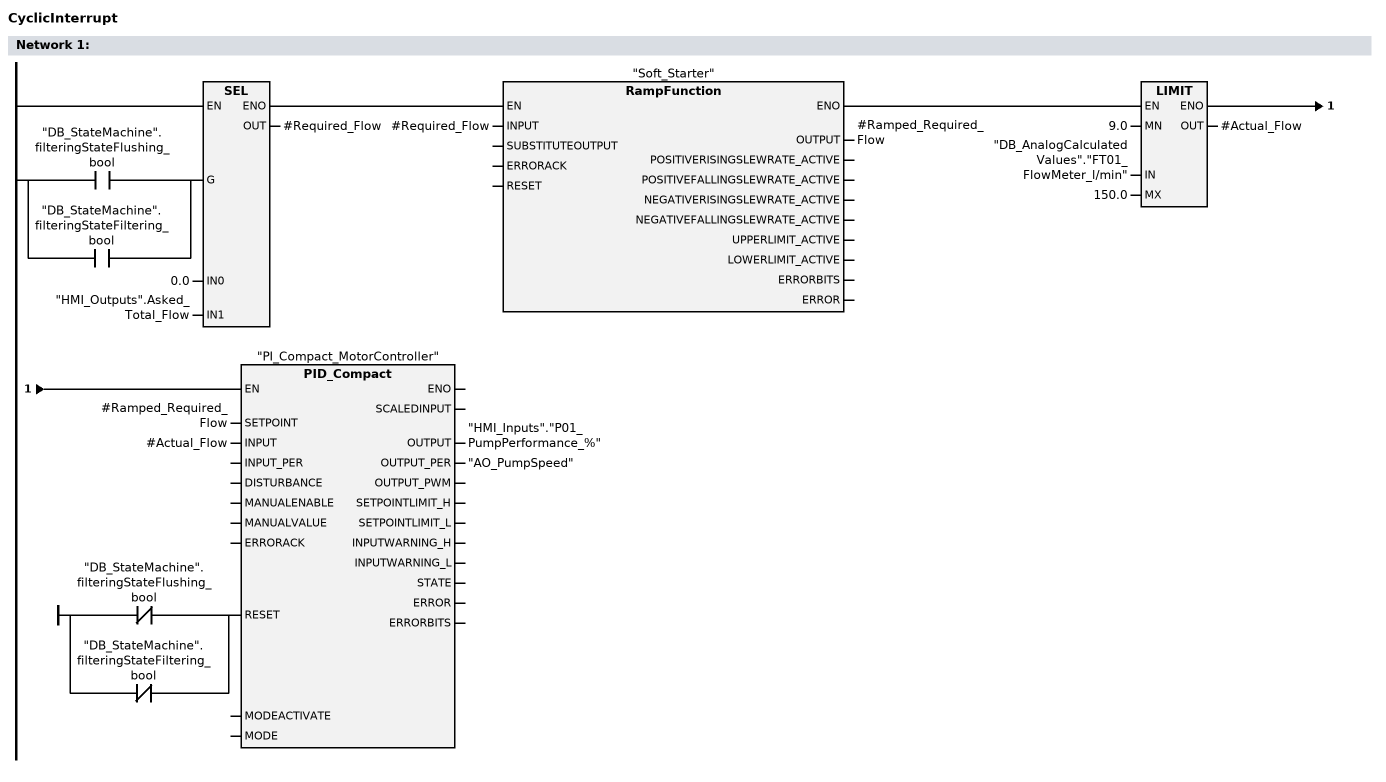
   // ENO of a box is taken as its EN; it also drops when the box reports an error
   #Required_Flow := SEL(G := "DB_StateMachine".filteringStateFlushing_bool OR "DB_StateMachine".filteringStateFiltering_bool, IN0 := 0.0, IN1 := "HMI_Outputs".Asked_Total_Flow);
   "Soft_Starter"(Input := #Required_Flow, Output => #Ramped_Required_Flow);   // RampFunction
   #Actual_Flow := LIMIT(MN := 9.0, IN := "DB_AnalogCalculatedValues"."FT01_FlowMeter_l/min", MX := 150.0);
   "PI_Compact_MotorController"(Setpoint := #Ramped_Required_Flow,   // PID_Compact
                           Input := #Actual_Flow,
                           Reset := NOT "DB_StateMachine".filteringStateFlushing_bool OR NOT "DB_StateMachine".filteringStateFiltering_bool,
                           Output => "HMI_Inputs"."P01_PumpPerformance_%",
                           Output_PER => "AO_PumpSpeed");
END_REGION
END_ORGANIZATION_BLOCK

ORGANIZATION_BLOCK "Startup"   // OB100, LAD, Startup
TITLE = "Complete Restart"
{ S7_Optimized_Access := 'TRUE' }
VERSION : 0.1
// Alapértékek beállítása.
   VAR_INPUT
      LostRetentive : Bool;   // True if retentive data are lost
      LostRTC : Bool;   // True if date and time are lost
   END_VAR
BEGIN

REGION Network 1 (SCL)
   // state machine init állapot beállítása
   "DB_StateMachine".actualState := "DB_StateMachine".initState;
   "DB_StateMachine".initState_bool := TRUE;

   //kimeneti értékek nullázása
   "DO_MotorStartSign" := false;
   "DO_TankFillValve" := false;
   "DO_OpenPermeateValve" := false;
   "DO_GreenLamp" := false;
   "DO_RedLamp" := false;
   "AO_PumpSpeed" := 0;

   //belső értékek nullázása
   "IT_Pump_DryRun_Fault" := false;
   "IT_Pump_Wrong_Valve_Setting_fault" := false;
   "PID_Reset_Value" := false;
   "IT_EStop_NOk" := false;
   "ErrorBit" := false;
   "Tag_7" := false;
   "Tag_8" := false;
   "Tag_9" := false;
   "Tag_10" := false;

   //state machine idle állapotra állítás
   //
   "DB_StateMachine".initState_bool := FALSE;
   IF NOT "DB_Errors&Warnings".error THEN

       "DB_StateMachine".actualState := 10;
       ;
   ELSE
       "DB_StateMachine".actualState := 900;
       ;
   END_IF;
END_REGION
END_ORGANIZATION_BLOCK